INTERFACE I_HMIBase EXTENDS	Base.I_BaseCyclic

PROPERTY P_BaseConfiguration : REFERENCE TO ST_BaseConfiguration
GET
END_GET
SET
END_SET
END_PROPERTY

PROPERTY P_BaseStatus : REFERENCE TO ST_BaseStatus
GET
END_GET
SET
END_SET
END_PROPERTY

PROPERTY P_Command : REFERENCE TO P_Command
GET
END_GET
SET
END_SET
END_PROPERTY

END_INTERFACE

(* stored: Version 1.1.0.1
   Itf I_HMIBase: Id {fa2c6f0a-b3ec-4ab4-a3a8-84ee08d4297f}
   Property P_BaseConfiguration: Id {0f638a4b-a0b4-422e-8d0b-f9a15f85558e}
   Get Get: Id {5010c0d8-f53e-496c-92ab-2ecaad598f06}
   Set Set: Id {d8dc285f-be01-4630-b74b-9ff5d51621a1}
   Property P_BaseStatus: Id {79051e6c-3bcf-465f-9dc4-8f7b3214282f}
   Get Get: Id {2ce5823d-012d-4729-8c36-1fbed4e87f02}
   Set Set: Id {ca104efe-1d79-4983-9fd3-f730833b67e1}
   Property P_Command: Id {9e6b1522-aff4-4b9e-ba8b-d9b6680509fe}
   Get Get: Id {ce938aff-42b5-41df-b89d-8680dd8f6d0c}
   Set Set: Id {7a801b8d-51d3-48ba-8183-7372f528efd4} *)
